TYPE COLOR : ARRAY[0..3] OF LREAL; END_TYPE

(* stored: Version 1.1.0.1
   DUT COLOR: Id {e53a2792-7c61-4707-9fb1-3deb3dbee952} *)
